// TIA Portal V21 export
DATA_BLOCK "ProductTransfer"   // DB310
// stored: AutoNumber false, InstanceOfName FB305, InstanceOfType FB
"FB305"
   // VAR_INPUT
   //    Enable : Bool;
   //    Disable : Bool;
   //    Fault : Bool;
   //    SecPulse : Bool;
   //    AlwaysTrue : Bool;
   //    StartConfirmationPopupSel : Bool;
   //    EndConfirmationPopupSel : Bool;
   //    WeightBasedSel : Bool;
   //    AdditionMethodSel : Bool;
   //    TransferTypeSel : Bool;
   //    TransferVesselPressureCheckSel : Bool;
   //    PressureReleaseSel : Bool;
   //    DelaytoEmptyLineSel : Bool;
   //    FlowSwitchCheckSel : Bool;
   //    TransfertoFMSel : Bool;
   //    RecBasedTransferSel : Bool;
   //    TemperatureControlSel : Bool;
   //    TransferMethodSel : Int;
   //    GasSel : Int;
   //    SetPressure : Real;
   //    SetVacuum : Real;
   //    SetQuantity : Real;
   //    SetSpeed : Real;
   //    ActualPressure : Real;
   //    ActualVacuum : Real;
   //    ActualQuantity : Real;
   //    ActualQuantityVessel : Real;
   //    FlowSwitchInput : Bool;
   //    FMHealthyInput : Bool;
   //    TemperatureReachedInput : Bool;
   //    PressureTol : Real;
   //    VacuumTol : Real;
   //    InflightQuantity : Real;
   //    VesselEmptyWeight : Real;
   //    DelaytoEmptyLine : Int;
   //    DelaytoReleaseTransferVesselPressure : Int;
   //    DelaytoReleasePressure : Int;
   //    DelaytoStartPump : Int;
   //    DelaytoOpenGasIn : Int;
   // END_VAR
   // VAR_OUTPUT
   //    AirValve : Bool;
   //    N2Valve : Bool;
   //    VacuumInValve : Bool;
   //    VacuumLineValves : Bool;
   //    LineValves : Bool;
   //    SuctionInValve : Bool;
   //    VesselOutletValve : Bool;
   //    RecirculationLineValves : Bool;
   //    FMInValve : Bool;
   //    PumpCmd : Bool;
   //    VacuumPumpCmd : Bool;
   //    StartConfirmationPopup : Bool;
   //    EndConfirmationPopup : Bool;
   //    ActualSpeed : Real;
   //    PrintTrigger : Bool;
   //    PrintWord : Int;
   //    PrintStatus : String[50];
   // END_VAR
   // VAR_IN_OUT
   //    Start : Bool;
   //    Stop : Bool;
   //    Reset : Bool;
   //    StartConfirmationAck : Bool;
   //    EndConfirmationAck : Bool;
   //    SpareBtn1 : Bool;
   //    SpareBtn2 : Bool;
   //    SpareBtn3 : Bool;
   //    Running : Bool;
   //    Selected : Bool;
   //    Paused : Bool;
   //    StartConfirmationPopupTemp : Bool;
   //    EndConfirmationPopupTemp : Bool;
   //    Started : Bool;
   //    Over : Bool;
   //    PumpBasedSelected : Bool;
   //    PressureBasedSelected : Bool;
   //    VacuumBasedSelected : Bool;
   //    StartDelaytoEmptyLine : Bool;
   //    StartDelaytoReleasePressure : Bool;
   //    SecondPopup : Bool;
   //    SecondPopupAck : Bool;
   //    PressureTolNeg : Real;
   //    VacuumTolNeg : Real;
   //    ActualSetQuantityCalc : Real;
   //    ActualSetQuantity : Real;
   // END_VAR
   // VAR
   //    ValveOnDelayPV : Int;
   //    ValveOffDelayPV : Int;
   //    PrintTriggerTemp : Bool;
   //    RE1 : Bool;
   //    RE2 : Bool;
   //    RE3 : Bool;
   //    RE4 : Bool;
   //    RE5 : Bool;
   //    RE6 : Bool;
   //    RE7 : Bool;
   //    PrintTriggerResetTimer { S7_SetPoint := 'True'} : TON_TIME;
   //    BtnResetTimer { S7_SetPoint := 'True'} : TON_TIME;
   //    TransferVesselPressureCheckDelay { S7_SetPoint := 'True'} : "FB103";
   //    PressureReleaseDelay { S7_SetPoint := 'True'} : "FB103";
   //    EmptyLineDelay { S7_SetPoint := 'True'} : "FB103";
   //    PumpOnDelayPv { S7_SetPoint := 'True'} : Int;
   // END_VAR
BEGIN
END_DATA_BLOCK
